FUNCTION_BLOCK RingTokenMemberHead (* Basic Function Block Type *)
  (* Standard: 61499-2 *)
  (* Version 0.2, 2003-12-04, JHC, Rockwell Automation, Renamed for better indexing. *)
  (* Version 0.1, 2002-11-05, JHC, Rockwell Automation, Corrected missing ST element in Algorithm REQ. *)
  (* Version 0.0, 2000-05-30, JHC, Rockwell Automation *)
  (* Compiler header: package fb.rt.cs725; *)
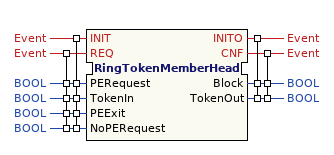
  EVENT_INPUT
    INIT WITH PERequest, TokenIn, PEExit, NoPERequest; (* Initialization Request *)
    REQ WITH PERequest, TokenIn, PEExit, NoPERequest; (* Normal Execution Request *)
  END_EVENT
  EVENT_OUTPUT
    INITO WITH Block, TokenOut; (* Initialization Confirm *)
    CNF WITH Block, TokenOut; (* Execution Confirmation *)
  END_EVENT
  VAR_INPUT
    PERequest : BOOL; (* Input event qualifier *)
    TokenIn : BOOL := true;
    PEExit : BOOL;
    NoPERequest : BOOL;
  END_VAR
  VAR_OUTPUT
    Block : BOOL; (* Output event qualifier *)
    TokenOut : BOOL := true;
  END_VAR
  VAR
    lastTokenIn : BOOL := true;
    lastPEExit : BOOL := 0;
    TokenChanged : BOOL := true;
  END_VAR
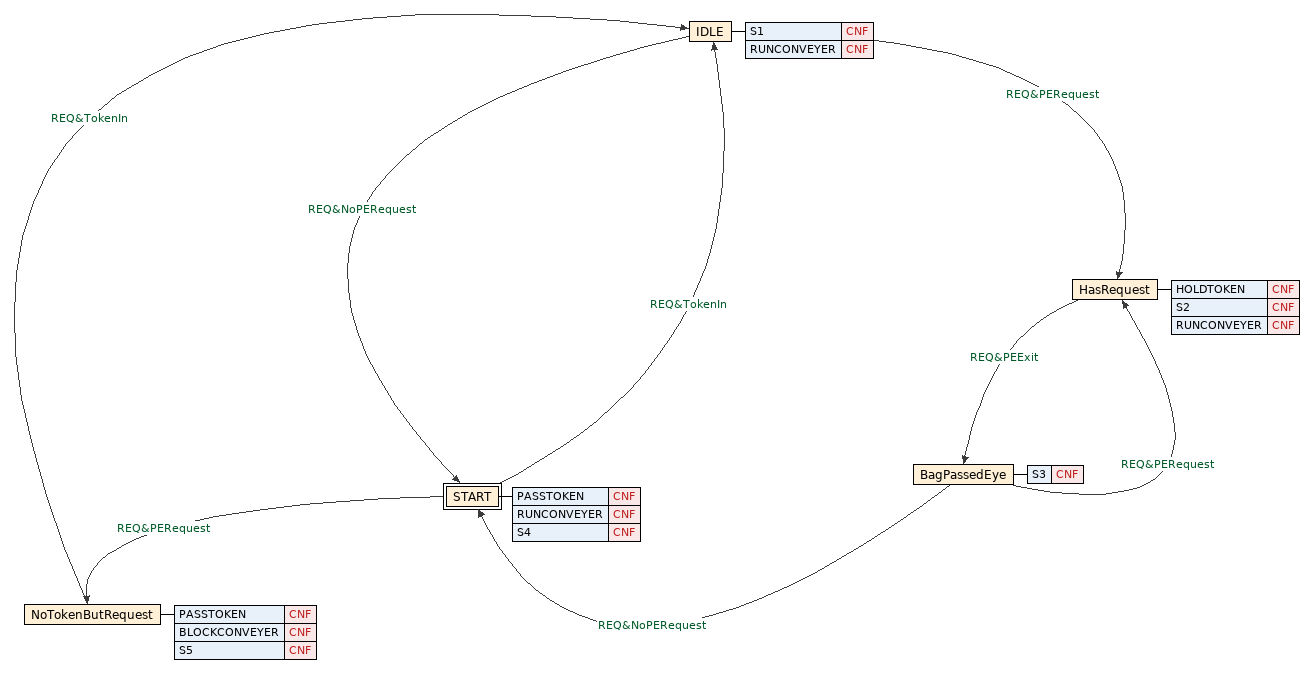
  EC_STATES
    START : PASSTOKEN -> CNF, RUNCONVEYER -> CNF, S4 -> CNF;
    IDLE : S1 -> CNF, RUNCONVEYER -> CNF;
    HasRequest : HOLDTOKEN -> CNF, S2 -> CNF, RUNCONVEYER -> CNF;
    BagPassedEye : S3 -> CNF;
    NoTokenButRequest : PASSTOKEN -> CNF, BLOCKCONVEYER -> CNF, S5 -> CNF;
  END_STATES
  EC_TRANSITIONS
    IDLE TO HasRequest := REQ&PERequest;
    HasRequest TO BagPassedEye := REQ&PEExit;
    START TO IDLE := REQ&TokenIn;
    BagPassedEye TO START := REQ&NoPERequest;
    BagPassedEye TO HasRequest := REQ&PERequest;
    START TO NoTokenButRequest := REQ&PERequest;
    NoTokenButRequest TO IDLE := REQ&TokenIn;
    IDLE TO START := REQ&NoPERequest;
  END_TRANSITIONS
  ALGORITHM INIT IN Java: (* Initialization algorithm *)
Block.value=false;
TokenOut.value=false;
System.out.println("init head, grant false, token true");
  END_ALGORITHM
  ALGORITHM REQ IN Java: (* Normally executed algorithm *)
System.out.println("3LastTokenIn, TokenIn, TokenOut:" + lastTokenIn.value + TokenIn.value + TokenOut.value);

if(lastTokenIn.value) {
if (TokenChanged.value) {
 if (!PERequest.value) {
  Block.value = false;
  TokenOut.value = false;
  System.out.println("Conv 3: I just got token, request is coming let bag go and keep token");
 } else {
  Block.value = false;
  TokenOut.value = true;
  System.out.println("Conv 3: I just got token, no request so run conveyer but let token go");
 }
} else {
 if (!PERequest.value) {
  System.out.println("Conv 3: I had token for a while, request here and bag passed eye, keep running conv and keep token");
  Block.value = false;
  TokenOut.value = false;
 } else {
  if (PEExit.value) {
   Block.value = false;
   TokenOut.value = true;
   System.out.println("Conv 3: I had token for a while, no requests and bag passed eye, let token go");
  } else {
   Block.value = false;
   TokenOut.value = false;
   System.out.println("Conv 3: I have token, no requests and bag not passed eye yet, keep token");
  }
 }
}
}

else {
    if (!PERequest.value) {
 Block.value = true;
TokenOut.value = true;
 System.out.println("Conv 3: No token, rquest here. Wait");
    }
else {
Block.value = false;
TokenOut.value = false;
System.out.println("Conv 3: No token no request");
}
}

if(lastTokenIn.value != TokenIn.value) {
    TokenChanged.value = true;
}
else {
    TokenChanged.value = false;
}
lastTokenIn.value = TokenIn.value;
  END_ALGORITHM
  ALGORITHM PASSTOKEN IN Java:
TokenOut.value=true;
//System.out.println("pass");
  END_ALGORITHM
  ALGORITHM HOLDTOKEN IN Java:
TokenOut.value=false;
//System.out.println("hold");
  END_ALGORITHM
  ALGORITHM BLOCKCONVEYER IN Java:
Block.value=true;
//System.out.println("block");
  END_ALGORITHM
  ALGORITHM RUNCONVEYER IN Java:
Block.value=false;
//System.out.println("run");
  END_ALGORITHM
  ALGORITHM S1 IN ST:
System.out.println("hSTATE 1");
  END_ALGORITHM
  ALGORITHM S2 IN ST:
System.out.println("hSTATE 2");
  END_ALGORITHM
  ALGORITHM S3 IN ST:
System.out.println("hSTATE 3");
  END_ALGORITHM
  ALGORITHM S4 IN ST:
System.out.println("hSTATE 4");
  END_ALGORITHM
  ALGORITHM S5 IN ST:
System.out.println("hSTATE 5");
  END_ALGORITHM
END_FUNCTION_BLOCK
